// Block: IPC_Com_Channel_LOG_PPRF

DATA_BLOCK IPC_Com_Channel_LOG_PPRF
VERSION : 0.1
   NON_RETAIN
   VAR
      RECEIVE : Struct
         ack : DInt;
         msg : IPC_Msg_Log_PPRF;
      END_STRUCT;
      SEND : Struct
         ack : DInt;
         msg : IPC_Msg_Log_PPRF;
      END_STRUCT;
   END_VAR

BEGIN
   // No initialization required
END_DATA_BLOCK
